// TIA Portal V19 export
VAR_GLOBAL   // PLC tag table "Default tag table_5"
END_VAR
